TYPE MyStruct :
STRUCT
  field1 : BOOL;
END_STRUCT
END_TYPE

(* stored: Version 1.0
   DUT MyStruct: Id {00000000-0000-0000-0000-000000000002} *)
